// Mitsubishi GX Works2 project: Project 1 14-05-2020   PLC: FX3G

PROGRAM MAIN
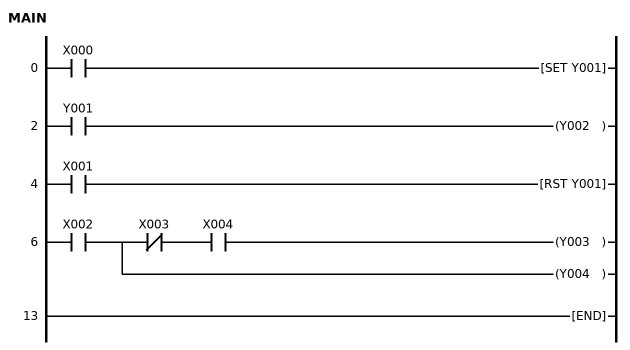
0     LD      X000
      SET     Y001
2     LD      Y001
      OUT     Y002
4     LD      X001
      RST     Y001
6     LD      X002
      MPS
      ANI     X003
      AND     X004
      OUT     Y003
      MPP
      OUT     Y004
13    END
END_PROGRAM
